TYPE T_TimeLog : STRING[15];
END_TYPE

(* stored: Version 1.1.0.1
   DUT T_TimeLog: Id {d6c954a7-3680-449f-a479-b0065ba4844e} *)
